INTERFACE ITF_TopElement2_HMI_Init EXTENDS ITF_BaseTopElement, ITF_TopElement2_HMI_Connector

END_INTERFACE

(* stored: Version 1.1.0.1
   Itf ITF_TopElement2_HMI_Init: Id {82bb1be1-4a35-0004-197a-49571a55df4d} *)
